TYPE U_BytesToReal :
UNION
    aBytes : ARRAY[0..3] OF BYTE;
    rValue : REAL;
END_UNION
END_TYPE

(* stored: Version 1.1.0.1
   DUT U_BytesToReal: Id {0d5c144b-f287-4c8f-b063-12160dda53e3} *)
